FUNCTION_BLOCK UDINT2TIME_2 (* Basic Function Block Type *)
  (* Standard: 61499-2 *)
  (* Version 0.0, 6/13/2026, Schneider Electric, Template *)
  PACKAGE SE.Nereda;
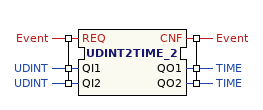
  EVENT_INPUT
    REQ WITH QI1, QI2; (* Normal Execution Request *)
  END_EVENT
  EVENT_OUTPUT
    CNF WITH QO1, QO2; (* Execution Confirmation *)
  END_EVENT
  VAR_INPUT
    QI1 : UDINT; (* Input event qualifier *)
    QI2 : UDINT;
  END_VAR
  VAR_OUTPUT
    QO1 : TIME; (* Output event qualifier *)
    QO2 : TIME;
  END_VAR
  VAR
    InQ1 : REAL;
    InQ2 : REAL;
  END_VAR
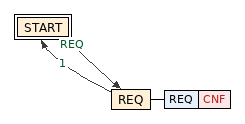
  EC_STATES
    START; (* Initial State *)
    REQ : REQ -> CNF; (* Normal execution *)
  END_STATES
  EC_TRANSITIONS
    START TO REQ := REQ;
    REQ TO START := 1;
  END_TRANSITIONS
  ALGORITHM REQ IN ST: (* Normally executed algorithm *)
;
InQ1 := UDINT_TO_REAL(QI1);
QO1 := REAL_TO_TIME(InQ1 * 1000);

InQ2 := UDINT_TO_REAL(QI2);
QO2 := REAL_TO_TIME(InQ2 * 1000);
  END_ALGORITHM
END_FUNCTION_BLOCK
